FUNCTION_BLOCK AX_PULSE (* Standard timer function block (pulse) - non-retriggerable *)
  (* Standard: 61499-2; Description: Copyright (c) 2023, 2024 HR Agrartechnik GmbH This program and the accompanying materials are made available under the terms of the Eclipse Public License 2.0 which is available at https://www.eclipse.org/legal/epl-2.0/ SPDX-License-Identifier: EPL-2.0 AX_PULSE -- Impulse forming FB with AX adapter interface Generate an Impulse with a given Time. This FB makes an Impulse of Duration PT on the Output Q. Non-retriggerable. *)
  (* Version 3.0, 2025-04-14, Patrick Aigner, changed package *)
  (* Version 1.1, 2024-04-23, Franz Höpfinger, HR Agrartechnik GmbH, Add a Reset to Timer FBs *)
  (* Version 1.0a, 2024-03-05, Franz Höpfinger, HR Agrartechnik GmbH, renamed to E_PULSE *)
  (* Version 1.0, 2023-08-21, Franz Höpfinger, HR Agrartechnik GmbH, initial implementation as E_IMPULSE *)
  PACKAGE adapter::events::unidirectional::timers;
  IMPORT eclipse4diac::core::TypeHash;
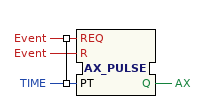
  EVENT_INPUT
    REQ WITH PT; (* Service Request *)
    R; (* Reset *)
  END_EVENT
  VAR_INPUT
    PT : TIME; (* Pulse time *)
  END_VAR
  PLUGS
    Q : adapter::types::unidirectional::AX; (* Timer output (AX adapter) *)
  END_PLUGS
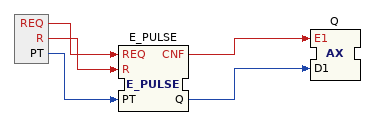
  FBS
    E_PULSE : iec61499::events::timers::E_PULSE;
  END_FBS
  EVENT_CONNECTIONS
    E_PULSE.CNF TO Q.E1;
    REQ TO E_PULSE.REQ;
    R TO E_PULSE.R;
  END_CONNECTIONS
  DATA_CONNECTIONS
    E_PULSE.Q TO Q.D1;
    PT TO E_PULSE.PT;
  END_CONNECTIONS
END_FUNCTION_BLOCK
